(* IEC 61131-3 sources: RL_MAR/experiments/comparison/llm4plc/results/Qwen-Qwen3.5-9B_20260506_150728/20260506_164036, 4 files *)

(* ---- generated_code_iteration_0.st ---- *)
START_ST
FUNCTION_BLOCK ChargingStationControl
VAR_INPUT
    EVConnected : BOOL;
    EVVoltage : REAL;
    EVCurrent : REAL;
    EVStateOfCharge : REAL;
    ChargingTimer : TIME;
END_VAR

VAR_OUTPUT
    EVCharging : BOOL;
END_VAR

VAR
    state : INT;
    VoltageOK : BOOL;
    CurrentOK : BOOL;
    SOCNotFull : BOOL;
    TimerOK : BOOL;
END_VAR

END_VAR

END_FUNCTION_BLOCK
END_ST

(* ---- generated_code_iteration_1.st ---- *)
START_REASON
The validation feedback indicates a CODESYS compiler error: "发现非预期的记号'END_VAR'" (Unexpected token 'END_VAR').

Analyzing the provided code:
1. The structure starts correctly with `FUNCTION_BLOCK` and `VAR_INPUT`.
2. The `VAR_INPUT` section ends with `END_VAR`.
3. The `VAR_OUTPUT` section ends with `END_VAR`.
4. The `VAR` section (local variables) is declared but **never closed**. It starts with `VAR` but lacks the corresponding `END_VAR`.
5. Immediately after the unclosed `VAR` section, the code has `END_VAR` again. This second `END_VAR` is interpreted as an attempt to close the `VAR` section, but since the previous `VAR` block was never explicitly closed (or the compiler expects the `VAR` block to be closed before the function block ends), this results in a syntax error. The compiler sees `END_VAR` where it expects the end of the variable list or the function block definition itself, but the structure is malformed because the `VAR` block is open.

The fix is simple: Add `END_VAR` after the `VAR` section (after `TimerOK : BOOL;`) to properly close the local variable declaration before the function block ends.
END_REASON

START_ST
FUNCTION_BLOCK ChargingStationControl
VAR_INPUT
    EVConnected : BOOL;
    EVVoltage : REAL;
    EVCurrent : REAL;
    EVStateOfCharge : REAL;
    ChargingTimer : TIME;
END_VAR

VAR_OUTPUT
    EVCharging : BOOL;
END_VAR

VAR
    state : INT;
    VoltageOK : BOOL;
    CurrentOK : BOOL;
    SOCNotFull : BOOL;
    TimerOK : BOOL;
END_VAR

END_FUNCTION_BLOCK
END_ST

(* ---- generated_code_iteration_2.st ---- *)
START_REASON
The previous error was caused by a character encoding issue. The feedback "gbk codec can't decode byte 0xa2" indicates that the code contains a non-ASCII character (likely a full-width comma or similar punctuation often introduced by copy-pasting from Chinese environments) that the CODESYS compiler cannot parse. Specifically, the comma after `TimerOK : BOOL;` in the `VAR` section is likely a full-width comma (，) instead of a standard ASCII comma (,).

Additionally, while the previous logic regarding `END_VAR` placement was sound, the encoding error prevents the code from being compiled at all. The fix requires replacing all potential non-standard punctuation with standard ASCII characters and ensuring the structure is clean.

The corrected code will:
1. Replace any full-width commas with standard ASCII commas.
2. Ensure all variable sections (`VAR_INPUT`, `VAR_OUTPUT`, `VAR`) are properly closed with `END_VAR`.
3. Maintain the `FUNCTION_BLOCK` structure.
END_REASON

START_ST
FUNCTION_BLOCK ChargingStationControl
VAR_INPUT
    EVConnected : BOOL;
    EVVoltage : REAL;
    EVCurrent : REAL;
    EVStateOfCharge : REAL;
    ChargingTimer : TIME;
END_VAR

VAR_OUTPUT
    EVCharging : BOOL;
END_VAR

VAR
    state : INT;
    VoltageOK : BOOL;
    CurrentOK : BOOL;
    SOCNotFull : BOOL;
    TimerOK : BOOL;
END_VAR

END_FUNCTION_BLOCK
END_ST

(* ---- generated_code_iteration_3.st ---- *)
START_REASON
The previous error "gbk codec can't decode byte 0x8c" indicates the presence of a non-ASCII character at position 429 in the file. In the GBK encoding scheme, byte 0x8c often corresponds to specific Chinese punctuation marks or characters that are not valid in standard IEC 61131-3 Structured Text (which requires ASCII).

Common culprits include:
1.  **Full-width commas (，)**: Often used in Chinese text, these look like standard commas but have different byte values.
2.  **Full-width colons (：)**: Similar to commas, these are frequently mistaken for standard colons.
3.  **Other invisible Unicode characters**: Sometimes copy-pasting from web interfaces introduces zero-width spaces or other invisible characters that break the parser.

The error occurs at position 429. Given the structure of a typical IEC 61131-3 function block, this position likely falls within the `VAR` section or the `END_VAR` statements. I need to ensure that every comma (`,`) and colon (`:`) used in the code is the standard ASCII version (0x2C and 0x3A respectively). I will regenerate the code ensuring strict ASCII compliance for all punctuation.

The corrected code will:
1.  Strictly use ASCII commas and colons.
2.  Ensure no hidden Unicode characters exist.
3.  Maintain the `FUNCTION_BLOCK` structure with correct `END_VAR` usage.
END_REASON

START_ST
FUNCTION_BLOCK ChargingStationControl
VAR_INPUT
    EVConnected : BOOL;
    EVVoltage : REAL;
    EVCurrent : REAL;
    EVStateOfCharge : REAL;
    ChargingTimer : TIME;
END_VAR

VAR_OUTPUT
    EVCharging : BOOL;
END_VAR

VAR
    state : INT;
    VoltageOK : BOOL;
    CurrentOK : BOOL;
    SOCNotFull : BOOL;
    TimerOK : BOOL;
END_VAR

END_FUNCTION_BLOCK
END_ST
